// TIA Portal V19 export
TYPE "Tel393In_PM"
// stored: Access Published
   STRUCT
      CU_ZSW1 : Struct   // Status word 1 for Control Unit
         sync : Bool;   // 1 = System time synchronized (SYNC)
         noAlarmPresent : Bool;   // 1 = No alarm present
         noFaultPresent : Bool;   // 1 = No fault present
         noSafetyMessagePresent : Bool;   // 1 = No safety message present
         slaveSignOfLifeBit0 : Bool;   // Slave sign of life bit 0
         slaveSignOfLifeBit1 : Bool;   // Slave sign of life bit 1
         slaveSignOfLifeBit2 : Bool;   // Slave sign of life bit 2
         slaveSignOfLifeBit3 : Bool;   // Slave sign of life bit 3
         reserved_Bit00 : Bool;   // Reserved
         reserved_Bit01 : Bool;   // Reserved
         reserved_Bit02 : Bool;   // Reserved
         faultPresent : Bool;   // 1 = Fault present
         reserved_Bit04 : Bool;   // Reserved
         reserved_Bit05 : Bool;   // Reserved
         reserved_Bit06 : Bool;   // Reserved
         alarmPresent : Bool;   // 1 = Alarm present
      END_STRUCT;
      E_DIGITAL : Struct   // Digital input (16 Bit)
         digitalInput0 : Bool;   // Digital input 0 (DI 0); p2081[8] = r0722.0
         digitalInput1 : Bool;   // Digital input 1 (DI 1); p2081[9] = r0722.1
         digitalInput2 : Bool;   // Digital input 2 (DI 2); p2081[10] = r0722.2
         digitalInput3 : Bool;   // Digital input 3 (DI 3); p2081[11] = r0722.3
         digitalInput4 : Bool;   // Digital input 4 (DI 4); p2081[12] = r0722.4
         digitalInput5 : Bool;   // Digital input 5 (DI 5); p2081[13] = r0722.5
         digitalInput6 : Bool;   // Digital input 6 (DI 6); p2081[14] = r0722.6
         digitalInput7 : Bool;   // Digital input 7 (DI 7); p2081[15] = r0722.7
         digitalInput8 : Bool;   // Digital input 8 (DI/DO 8); p2081[0] = r0722.8
         digitalInput9 : Bool;   // Digital input 9 (DI/DO 9); p2081[1] = r0722.9
         digitalInput10 : Bool;   // Digital input 10 (DI/DO 10); p2081[2] = r0722.10
         digitalInput11 : Bool;   // Digital input 11 (DI/DO 11); p2081[3] = r0722.11
         digitalInput12 : Bool;   // Digital input 12 (DI/DO 12); p2081[4] = r0722.12
         digitalInput13 : Bool;   // Digital input 13 (DI/DO 13); p2081[5] = r0722.13
         digitalInput14 : Bool;   // Digital input 14 (DI/DO 14); p2081[6] = r0722.14
         digitalInput15 : Bool;   // Digital input 15 (DI/DO 15); p2081[7] = r0722.15
      END_STRUCT;
      E_DIGITAL_1 : Struct   // Digital input (16 Bit)
         digitalInput16 : Bool;   // Digital input 16 (DI 16); p2083[8] = r0722.16
         digitalInput17 : Bool;   // Digital input 17 (DI 17); p2083[9] = r0722.17
         digitalInput18 : Bool;   // Digital input 18 (DI 18); p2083[10] = r0722.18
         digitalInput19 : Bool;   // Digital input 19 (DI 19); p2083[11] = r0722.19
         digitalInput20 : Bool;   // Digital input 20 (DI 20); p2083[12] = r0722.20
         digitalInput21 : Bool;   // Digital input 21 (DI 21); p2083[13] = r0722.21
         digitalInput22 : Bool;   // Digital input 22 (DI 22); p2083[14] = r0722.22
         reserved_Bit15 : Bool;   // Reserved
         Axis1_PathTestReq : Bool;   // Set p2083[0] with Axis r7923.0
         Axis1_PathTestRunning : Bool;   // Set p2083[1] with Axis r7923.12
         Axis2_PathTestReq : Bool;   // Set p2083[2] with Axis r7923.0
         Axis2_PathTestRunning : Bool;   // Set p2083[3] with Axis r7923.12
         Axis3_PathTestReq : Bool;   // Set p2083[4] with Axis r7923.0
         Axis3_PathTestRunning : Bool;   // Set p2083[5] with Axis r7923.12
         Axis4_PathTestReq : Bool;   // Set p2083[6] with Axis r7923.0
         Axis4_PathTestRunning : Bool;   // Set p2083[7] with Axis r7923.12
      END_STRUCT;
      MT_ZSW : Struct   // Measuring probe status word
         digitalInputProbe1 : Bool;   // Digital input display
         digitalInputProbe2 : Bool;   // Digital input display
         digitalInputProbe3 : Bool;   // Digital input display
         digitalInputProbe4 : Bool;   // Digital input display
         digitalInputProbe5 : Bool;   // Digital input display
         digitalInputProbe6 : Bool;   // Digital input display
         digitalInputProbe7 : Bool;   // Digital input display
         digitalInputProbe8 : Bool;   // Digital input display
         subSamplingProbe1 : Bool;   // Not yet carried out
         subSamplingProbe2 : Bool;   // Not yet carried out
         subSamplingProbe3 : Bool;   // Not yet carried out
         subSamplingProbe4 : Bool;   // Not yet carried out
         subSamplingProbe5 : Bool;   // Not yet carried out
         subSamplingProbe6 : Bool;   // Not yet carried out
         subSamplingProbe7 : Bool;   // Not yet carried out
         subSamplingProbe8 : Bool;   // Not yet carried out
      END_STRUCT;
      MT1_ZS_F : Word;   // Measuring probe 1 measuring time falling edge
      MT1_ZS_S : Word;   // Measuring probe 1 measuring time rising edge
      MT2_ZS_F : Word;   // Measuring probe 2 measuring time falling edge
      MT2_ZS_S : Word;   // Measuring probe 2 measuring time rising edge
      MT3_ZS_F : Word;   // Measuring probe 3 measuring time falling edge
      MT3_ZS_S : Word;   // Measuring probe 3 measuring time rising edge
      MT4_ZS_F : Word;   // Measuring probe 4 measuring time falling edge
      MT4_ZS_S : Word;   // Measuring probe 4 measuring time rising edge
      MT5_ZS_F : Word;   // Measuring probe 5 measuring time falling edge
      MT5_ZS_S : Word;   // Measuring probe 5 measuring time rising edge
      MT6_ZS_F : Word;   // Measuring probe 6 measuring time falling edge
      MT6_ZS_S : Word;   // Measuring probe 6 measuring time rising edge
      MT7_ZS_F : Word;   // Measuring probe 7 measuring time falling edge
      MT7_ZS_S : Word;   // Measuring probe 7 measuring time rising edge
      MT8_ZS_F : Word;   // Measuring probe 8 measuring time falling edge
      MT8_ZS_S : Word;   // Measuring probe 8 measuring time rising edge
      E_ANALOG : Word;   // Analog inputs
   END_STRUCT;
END_TYPE
